FUNCTION_BLOCK TFAggiuntaSupportoManuale
VAR_INPUT
	WorkArea : POINTER TO ARRAY [1..MAXAREA] OF TFMachinePalletizer_WorkArea;
	WorkAreaState : POINTER TO ARRAY [1..MAXAREA] OF TFMachinePalletizer_WorkAreaState;
	WorkAreaNumber : UINT; //Numero postazione
	Forming : POINTER TO ARRAY [1..MAXFORMING] OF TFMachinePalletizer_FormingForSlab;
	Pallet : POINTER TO ARRAY [1..MAXPALLET] OF TFMachinePalletizer_Pallet;
	Layer : POINTER TO ARRAY [1..MAXLAYER] OF TFMachinePalletizer_Layer;
	ProgressiveNrWA : POINTER TO UDINT;
	CodicePostazione : INT;
	IndiceFormaturaPostazione : INT;
	AbilitaAssegnazioneCodicePiazzoleConPaccoSuRibaltino : BOOL;
	InserisciNuovoPallet : BOOL;
	PH_Presenza : bool;// ARRAY[1..MAXAREA] OF BOOL;
END_VAR
VAR_OUTPUT
END_VAR
VAR
	PHPostazioniUPTrig 			: ARRAY[1..MAXAREA] OF BOOL;
	PHPostazioniDOWNTrig 		: ARRAY[1..MAXAREA] OF BOOL;
	UltimaFormaturaAssegnata 	: INT;
	UltimaPostazioneCancellata 	: UINT;
	UltimaPostazioneCreata 		: UINT;
	Zone : INT;
	ar: INT;
	cod : INT;
	FormaturaZona : ARRAY[1..MAXFORMINGCODE] OF INT;
	FormaturePresenti : ARRAY[1..MAXFORMING] OF INT;
	DoppiaFormaturaAttiva :BOOL;
	CodiceInFormaturaMem : INT;
	NumCodiciInFormaturaAttiviPerZona : UINT;	

END_VAR

InserisciNuovoPallet:= FALSE;
//Fronte salita
IF PH_Presenza AND NOT PHPostazioniUPTrig[WorkAreaNumber] THEN
	PHPostazioniUPTrig[WorkAreaNumber] := TRUE;
	UltimaPostazioneCreata := WorkAreaNumber;
ELSIF NOT PH_Presenza AND PHPostazioniUPTrig[WorkAreaNumber] THEN
	PHPostazioniUPTrig[WorkAreaNumber] := FALSE;
END_IF
//Fronte discesa
//Pulisco la postazione
IF NOT PH_Presenza AND NOT PHPostazioniDOWNTrig[WorkAreaNumber] THEN
	PHPostazioniDOWNTrig[WorkAreaNumber] := TRUE;
	UltimaPostazioneCancellata := WorkAreaNumber;
	IF WorkAreaState^[WorkAreaNumber].State >= WORKAREA_STATE_OCCUPIED_WORKING THEN
		TFClearWorkAreaArray(WorkArea,WorkAreaState,WorkAreaNumber);
	END_IF
	
	IF WorkAreaNumber = Mission.PPlace THEN
	//Modificacion borrar datos piking Al sacar el soporte
	MEMSET(destAddr := ADR(HMi_DimensionesPiezasWorkAreaDeposito),fillByte := 0 , n := SIZEOF(HMi_DimensionesPiezasWorkAreaDeposito));
	END_IF
	
ELSIF PH_Presenza AND PHPostazioniDOWNTrig[WorkAreaNumber] THEN
	PHPostazioniDOWNTrig[WorkAreaNumber] := FALSE;
END_IF

//Verifico se è stato inserito il nuovo codice del pallet
IF (WorkAreaState^[WorkAreaNumber].Code > 0 OR PHPostazioniUPTrig[WorkAreaNumber]) AND (WorkArea^[WorkAreaNumber].Enable = 1 AND WorkAreaState^[WorkAreaNumber].State < WORKAREA_STATE_OCCUPIED_WORKING AND WorkAreaState^[WorkAreaNumber].State <> 1) THEN
	InserisciNuovoPallet := TRUE;
END_IF

IF InserisciNuovoPallet AND WorkAreaState^[WorkAreaNumber].State < WORKAREA_STATE_OCCUPIED_WORKING THEN	
	
	WorkAreaState^[WorkAreaNumber].Taped := -1;
	WorkAreaState^[WorkAreaNumber].LGV_ReqAbort := FALSE;
	
	WorkAreaState^[WorkAreaNumber].Supporto := Forming^[1].Pallet;
	WorkAreaState^[WorkAreaNumber].F := 1;
	WorkAreaState^[WorkAreaNumber].ID 	:= ProgressiveNrWA^;
	ProgressiveNrWA^ := ProgressiveNrWA^ + 1;
	WorkAreaState^[WorkAreaNumber].P 	:= 0;
	WorkAreaState^[WorkAreaNumber].Slow := 1;
	WorkAreaState^[WorkAreaNumber].LGVAttr := Forming^[WorkAreaState^[WorkAreaNumber].F].LGVAttr;
	WorkAreaState^[WorkAreaNumber].State := WORKAREA_STATE_OCCUPIED_WORKING;
	
	InserisciNuovoPallet := FALSE;

ELSIF InserisciNuovoPallet AND WorkAreaState^[WorkAreaNumber].State < WORKAREA_STATE_OCCUPIED_WORKING AND FALSE THEN
	
	//Se la postazione ha codice fisso, lo assegno!
	IF CodicePostazione = 0 AND WorkAreaCodiciFissi[WorkAreaNumber] > 0 THEN
		CodicePostazione := WorkAreaCodiciFissi[WorkAreaNumber];
	END_IF

	(* Cerco Formatura *)
	IndiceFormaturaPostazione := 0;
	IndiceFormaturaPostazione := TFPalletizerGetFormingFromCodeSlab(Forming,CodicePostazione);
	//Assegno la formatura successivamanete nel WAManager
	IF IndiceFormaturaPostazione < 1 THEN
		IndiceFormaturaPostazione := 0;
		//Valuto la zona della postazione e ricavo la formatura in base alla zona di appartenenza	
	
		FOR cod:=1 TO MAXFORMINGCODE DO
			FormaturaZona[cod] := 0;
		END_FOR
		DoppiaFormaturaAttiva := FALSE;
		CodiceInFormaturaMem := 0;
		NumCodiciInFormaturaAttiviPerZona := 0;
		FOR zone:=1 TO MAXZONE DO
			FOR ar:=1 TO MAXAREA DO
				(* Verifico se la WorkArea appartiena ad una Zona *)
				IF WorkAreaZone.Zone[zone].WorkArea[ar] = WorkAreaNumber THEN
					FOR cod:=1 TO MAXFORMINGCODE DO
						IF FormaturaZona[cod] > 0 THEN
							DoppiaFormaturaAttiva := TRUE;
						END_IF
						FormaturaZona[cod] := TFPalletizerGetFormingFromCodeSlab(Forming,WorkAreaZone.Zone[zone].Code[cod]);
						IF WorkAreaZone.Zone[zone].Code[cod] <> CodiceInFormaturaMem  THEN//Memorizzo se ho un codice 
							NumCodiciInFormaturaAttiviPerZona := NumCodiciInFormaturaAttiviPerZona+1;
							CodiceInFormaturaMem := WorkAreaZone.Zone[zone].Code[cod];
						END_IF
					END_FOR
					EXIT;//Esco e vado a valutare le formature
				END_IF
			END_FOR
		END_FOR	
		FOR ar:=1 TO 4 DO
			FormaturePresenti[ar] := 0;
		END_FOR
		FOR ar:=1 TO MAXFORMINGCODE DO
		
			CASE FormaturaZona[ar] OF
				1:
					FormaturePresenti[1] := FormaturePresenti[1]+1; 	
				2:
					FormaturePresenti[2] := FormaturePresenti[2]+1;
				3:
					FormaturePresenti[3] := FormaturePresenti[3]+1;
				4:
					FormaturePresenti[4] := FormaturePresenti[4] +1;
			ELSE
				IndiceFormaturaPostazione := 0;			
			END_CASE				
		END_FOR
		//Cerco se nella zona ci sono + formature presenti, se è così codice formatura = 0, in modo che la macchina lo assagne in base alle esigenze
		//Altrimenti se solo una formatura è presente gli assegno quella!			
		IF FormaturePresenti[1] >= 1 THEN
			IF FormaturePresenti[2] >= 1 OR FormaturePresenti[3] >= 1 OR FormaturePresenti[4] >= 1 OR DoppiaFormaturaAttiva THEN
				IndiceFormaturaPostazione := 0;
			ELSE
				IndiceFormaturaPostazione := 1;
				IF NumCodiciInFormaturaAttiviPerZona = 1 THEN
					 CodicePostazione := CodiceInFormaturaMem;
				END_IF
			END_IF		
		ELSIF FormaturePresenti[2] >= 1 THEN
			IF FormaturePresenti[1] >= 1 OR FormaturePresenti[3] >= 1 OR FormaturePresenti[4] >= 1 OR DoppiaFormaturaAttiva THEN
				IndiceFormaturaPostazione := 0;
			ELSE
				IndiceFormaturaPostazione := 2;
				IF NumCodiciInFormaturaAttiviPerZona = 1 THEN
					 CodicePostazione := CodiceInFormaturaMem;
				END_IF
			END_IF		
		ELSIF FormaturePresenti[3] >= 1 THEN
			IF FormaturePresenti[2] >= 1 OR FormaturePresenti[1] >= 1 OR FormaturePresenti[4] >= 1 OR DoppiaFormaturaAttiva THEN
				IndiceFormaturaPostazione := 0;
			ELSE
				IndiceFormaturaPostazione := 3;
				IF NumCodiciInFormaturaAttiviPerZona = 1 THEN
					 CodicePostazione := CodiceInFormaturaMem;
				END_IF
			END_IF		
		ELSIF FormaturePresenti[4] >= 1 THEN
			IF FormaturePresenti[2] >= 1 OR FormaturePresenti[3] >= 1 OR FormaturePresenti[1] >= 1 OR DoppiaFormaturaAttiva THEN
				IndiceFormaturaPostazione := 0;
			ELSE
				IndiceFormaturaPostazione := 4;
				IF NumCodiciInFormaturaAttiviPerZona = 1 THEN
					 CodicePostazione := CodiceInFormaturaMem;
				END_IF
			END_IF		
		END_IF
	END_IF
	
	WorkAreaState^[WorkAreaNumber].Taped := -1;
	WorkAreaState^[WorkAreaNumber].LGV_ReqAbort := FALSE;
	IF AbilitaAssegnazioneCodicePiazzoleConPaccoSuRibaltino AND CodicePostazione = 0 THEN
		WorkAreaState^[WorkAreaNumber].Code := 0;
		WorkAreaState^[WorkAreaNumber].Initialize := TRUE;
	ELSE
		WorkAreaState^[WorkAreaNumber].Code := CodicePostazione;
		WorkAreaState^[WorkAreaNumber].Initialize := FALSE;
	END_IF
	WorkAreaState^[WorkAreaNumber].Supporto := Forming^[IndiceFormaturaPostazione].Pallet;
	WorkAreaState^[WorkAreaNumber].F := IndiceFormaturaPostazione;
	
	WorkAreaState^[WorkAreaNumber].ID := ProgressiveNrWA^;
	ProgressiveNrWA^ := ProgressiveNrWA^ + 1;
	WorkAreaState^[WorkAreaNumber].P := 0;
	WorkAreaState^[WorkAreaNumber].Slow := 1;
	WorkAreaState^[WorkAreaNumber].LGVAttr := Forming^[WorkAreaState^[WorkAreaNumber].F].LGVAttr;
	WorkAreaState^[WorkAreaNumber].State := WORKAREA_STATE_OCCUPIED_WORKING;

	InserisciNuovoPallet := FALSE;
END_IF

END_FUNCTION_BLOCK

(* stored: Version 1.1.0.1, ProductVersion 3.1.4024.11
   POU TFAggiuntaSupportoManuale: Id {4b97a81a-5c2e-4454-a72d-363c5ed22724}, SpecialFunc None *)
